{attribute 'GeneratedUsingTerminal: EK1122-0000-0018'}
{attribute addProperty BoxType "EK1122-0000-0018"}
{attribute addProperty Id "Beckhoff_ELM3xxx_0030sub_EK1100EK1100_1FC0878B2"}
{attribute addProperty CRC "2511433776"}
{attribute addProperty Size "2"}
TYPE Beckhoff_ELM3xxx_0030EK1122_95B17030 EXTENDS EK1122_1FC0878B :
STRUCT
	{attribute addProperty Name "Beckhoff_ELM3xxx_0030sub_EK1100"}
	{attribute addProperty PreviousPort "Beckhoff ELM3xxx-0030EK1122 : D"}
	Beckhoff_ELM3xxx_0030sub_EK1100 : EK1100_1FC0878B;
END_STRUCT
END_TYPE

(* stored: Version 1.2.0.0, ProductVersion 3.1.4024.9
   DUT Beckhoff_ELM3xxx_0030EK1122_95B17030: Id {db516bde-120a-4a58-b91b-2933da988c48} *)
